(* CODESYS project Esp32ModbusTCP.library
   Company: EvisLab Automation
   DefaultNamespace: ESP32
   Version: 1.0.0.1
   Placeholder: ESP32 ModbusTCP
   Author: Evis Vasiu
   Description: Write coils FC-15: 0 - 39 (connected to Digital Outputs)
      Read inputs FC-02: 100 - 139 (connected to Digital Inputs)
      Write Holding Registers FC-16: 200 - 239 (connected to Analog Output (DAC), PWM pins)
      Read Input Registers FC-04: 300 - 339 (connected to Analog Inputs)
      
      Port: 502
   Title: ESP32 ModbusTCP

Project tree, tasks and I/O mapping:
  libraries: Tc2_BABasic, * (Beckhoff Automation GmbH); Tc2_ModbusSrv, 3.3.2.0 (Beckhoff Automation GmbH); Tc2_Standard, * (Beckhoff Automation GmbH); Tc2_System, * (Beckhoff Automation GmbH); Tc3_Module, * (Beckhoff Automation GmbH)
  DUTs/
    data type Esp32Discrete
    data type Esp32Registers
  GVLs/
  POUs/
    function block FB_Esp32ModbusTCP [ST]
  Version/
    global variables Global_Version
*)

// DUTs/Esp32Discrete
TYPE Esp32Discrete :
STRUCT
	pin0 : BIT;
	pin1 : BIT;
	pin2 : BIT;
	pin3 : BIT;
	pin4 : BIT;
	pin5 : BIT;
	pin6 : BIT;
	pin7 : BIT;
	pin8 : BIT;
	pin9 : BIT;
	pin10: BIT;
	pin11: BIT;
	pin12: BIT;
	pin13: BIT;
	pin14: BIT;
	pin15: BIT;
	pin16: BIT;
	pin17: BIT;
	pin18: BIT;
	pin19: BIT;
	pin20: BIT;
	pin21: BIT;
	pin22: BIT;
	pin23: BIT;
	pin24: BIT;
	pin25: BIT;
	pin26: BIT;
	pin27: BIT;
	pin28: BIT;
	pin29: BIT;
	pin30: BIT;
	pin31: BIT;
	pin32: BIT;
	pin33: BIT;
	pin34: BIT;
	pin35: BIT;
	pin36: BIT;
	pin37: BIT;
	pin38: BIT;
	pin39: BIT;

END_STRUCT
END_TYPE

// DUTs/Esp32Registers
TYPE Esp32Registers :
STRUCT
	pin0 : INT;
	pin1 : INT;
	pin2 : INT;
	pin3 : INT;
	pin4 : INT;
	pin5 : INT;
	pin6 : INT;
	pin7 : INT;
	pin8 : INT;
	pin9 : INT;
	pin10: INT;
	pin11: INT;
	pin12: INT;
	pin13: INT;
	pin14: INT;
	pin15: INT;
	pin16: INT;
	pin17: INT;
	pin18: INT;
	pin19: INT;
	pin20: INT;
	pin21: INT;
	pin22: INT;
	pin23: INT;
	pin24: INT;
	pin25: INT;
	pin26: INT;
	pin27: INT;
	pin28: INT;
	pin29: INT;
	pin30: INT;
	pin31: INT;
	pin32: INT;
	pin33: INT;
	pin34: INT;
	pin35: INT;
	pin36: INT;
	pin37: INT;
	pin38: INT;
	pin39: INT;

END_STRUCT
END_TYPE

// Version/Global_Version
{attribute 'TcGenerated'}
{attribute 'no-analysis'}
{attribute 'linkalways'}
// This function has been automatically generated from the project information.
VAR_GLOBAL CONSTANT
	{attribute 'const_non_replaced'}
	stLibVersion_ESP32_ModbusTCP : ST_LibVersion := (iMajor := 1, iMinor := 0, iBuild := 0, iRevision := 1, nFlags := 0, sVersion := '1.0.0.1');
END_VAR

// POUs/FB_Esp32ModbusTCP
FUNCTION_BLOCK FB_Esp32ModbusTCP
VAR_INPUT
	IP      : STRING(15);
	WriteCoils : Esp32Discrete;
	WriteHoldingRegisters : Esp32Registers;
END_VAR

VAR_OUTPUT
	ReadDiscreteInputs : Esp32Discrete;
	ReadInputRegisters : Esp32Registers;	
END_VAR

VAR
	
	fbMBWriteCoils : FB_MBWriteCoils;
	fbMBReadInputs : FB_MBReadInputs;
	fbMBWriteRegs : FB_MBWriteRegs;
	fbMBReadInputRegs : FB_MBReadInputRegs ;
	
	count : BYTE := 0;

END_VAR


	count := count +1 ;
	IF count > 3 THEN
		count := 0;
	END_IF

CASE count OF
	0:
	fbMBWriteCoils (
	sIPAddr := IP,
	nTCPPort := 502, 
	nUnitID := 16#FF,
	nQuantity := 40,
	nMBAddr   := 0,
	cbLength  := SIZEOF(WriteCoils),
	pSrcAddr  := ADR(WriteCoils),
	bExecute:= NOT fbMBWriteCoils.bBusy AND NOT fbMBReadInputs.bBusy AND NOT fbMBWriteRegs.bBusy AND NOT fbMBReadInputRegs.bBusy,
	tTimeout := T#2S);
	
	1:
	fbMBReadInputs (
	sIPAddr := IP,
	nTCPPort := 502, 
	nUnitID := 16#FF,
	nQuantity := 40,
	nMBAddr   := 100,
	cbLength  := SIZEOF(ReadDiscreteInputs),
	pDestAddr := ADR(ReadDiscreteInputs),
	bExecute:= NOT fbMBWriteCoils.bBusy AND NOT fbMBReadInputs.bBusy AND NOT fbMBWriteRegs.bBusy AND NOT fbMBReadInputRegs.bBusy,
	tTimeout := T#2S);
	
	2:
	fbMBWriteRegs (
	sIPAddr := IP,
	nTCPPort := 502, 
	nUnitID := 16#FF,
	nQuantity := 40,
	nMBAddr   := 200,
	cbLength  := SIZEOF(WriteHoldingRegisters),
	pSrcAddr   := ADR(WriteHoldingRegisters),
	bExecute:= NOT fbMBWriteCoils.bBusy AND NOT fbMBReadInputs.bBusy AND NOT fbMBWriteRegs.bBusy AND NOT fbMBReadInputRegs.bBusy,
	tTimeout := T#2S);
	
	3:
	fbMBReadInputRegs (
	sIPAddr := IP,
	nTCPPort := 502, 
	nUnitID := 16#FF,
	nQuantity := 40,
	nMBAddr   := 300,
	cbLength  := SIZEOF(ReadInputRegisters),
	pDestAddr := ADR(ReadInputRegisters),
	bExecute:= NOT fbMBWriteCoils.bBusy AND NOT fbMBReadInputs.bBusy AND NOT fbMBWriteRegs.bBusy AND NOT fbMBReadInputRegs.bBusy,
	tTimeout := T#2S);
	
END_CASE

END_FUNCTION_BLOCK
